// TIA Portal V20 export
// export: Created 2025-12-01T14:57:05.2078654Z, ExportSetting None, DisplayName Totally Integrated Automation Portal, DisplayVersion V20 Update 3, DisplayName TIA Portal Openness, DisplayVersion V20 Update 3, DisplayName TIA Portal Version Control Interface, DisplayVersion V20 Update 3, DisplayName STEP 7 Professional, DisplayVersion V20 Update 3, DisplayName STEP 7 Safety, DisplayVersion V20 Update 2, DisplayName WinCC Basic/Comfort/Advanced, DisplayVersion V20 Update 3, DisplayName WinCC Professional, DisplayVersion V20 Update 3, DisplayName WinCC Unified, DisplayVersion V20 Update 3
FUNCTION "FC836_GestorEstadoMaquina" : Void   // FC836, LAD
TITLE = Tracking Envio Solo del Estado de una Maquina
{ S7_Optimized_Access := 'FALSE' }
AUTHOR : TRACKING
NAME : 20130322
VERSION : 3.0
// stored: AutoNumber false, SetENOAutomatically false
   VAR_INPUT
      NumMaquina : UInt;   // Numero de la Maquina
      Automatico : Bool;   // Automatico / Manual
      Marcha : Bool;   // Marcha / Paro
      Error : Bool;   // Error
      CodigoError : UDInt;   // Codigo de Error
   END_VAR
   VAR_TEMP
      Maquina : UInt;
      CodigoErrorMaquina : UDInt;
   END_VAR
BEGIN

NETWORK
TITLE = Inicializar
//////////////////////////////////////////////////////////////////////////
// --- Inicializar las Variables

      L     #NumMaquina;  // Numero de Maquina
      T     #Maquina;



NETWORK
TITLE = Guardar Status
//////////////////////////////////////////////////////////////////////////
//////////////////////////////////////////////////////////////////////////
//////////////////////////////////////////////////////////////////////////
// --- Estado de Automatico - Manual
      SET;
      A     #Automatico;
      =     "DB840_Emision".DispoMaquina[#Maquina].Protocolo.Automatico;

      SET;
      AN    #Automatico;
      =     "DB840_Emision".DispoMaquina[#Maquina].Protocolo.Manual;


//////////////////////////////////////////////////////////////////////////
//////////////////////////////////////////////////////////////////////////
//////////////////////////////////////////////////////////////////////////
// --- Estado de Marcha - Paro - Error
      SET;
      A     #Marcha;
      =     "DB840_Emision".DispoMaquina[#Maquina].Protocolo.Marcha;

      SET;
      AN    #Marcha;
      =     "DB840_Emision".DispoMaquina[#Maquina].Protocolo.Paro;

      SET;
      A     #Error;
      =     "DB840_Emision".DispoMaquina[#Maquina].Protocolo.Error;


//////////////////////////////////////////////////////////////////////////
//////////////////////////////////////////////////////////////////////////
//////////////////////////////////////////////////////////////////////////
// ---  Guardo Error  Depediendo si hay Error
      SET;
      AN    #Error;
      JC    SinError_EnMaquina;
      JU    ConError_EnMaquina;


//////////////////////////////////////////////////////////////////////////
// --- Sin Error
SinError_EnMaquina:NOP   0;
      L     0;
      T     "DB840_Emision".DispoMaquina[#Maquina].Error;
      T     "DB861_FIFO_Errores".Maquinas[#Maquina];

      BE;


//////////////////////////////////////////////////////////////////////////
// --- Sin Error
ConError_EnMaquina:NOP   0;
      L     #CodigoError;
      T     #CodigoErrorMaquina;
      T     "DB861_FIFO_Errores".Maquinas[#Maquina];

      L     #CodigoError;  // Maquina
      T     "DB840_Emision".DispoMaquina[#Maquina].Error;

      BE;


END_FUNCTION
